FUNCTION_BLOCK Cylinder 
VAR_INPUT
END_VAR
VAR_OUTPUT
	bExtended : BOOL;
	bExtend : BOOL;
END_VAR
VAR
	fbExtendedSignal : BoolIn;
	fbExtend : BoolOut;
END_VAR

bExtended := fbExtendedSignal.getValue;
bExtend := fbExtend.getValue;

METHOD Extend : BOOL
VAR_INPUT
END_VAR
fbExtend.setValue := TRUE;
END_METHOD

PROPERTY getExtend : I_StepCondition
GET
getExtend := fbExtend;
END_GET
END_PROPERTY

METHOD Retract : BOOL
VAR_INPUT
END_VAR
fbExtend.setValue := FALSE;
END_METHOD

END_FUNCTION_BLOCK

(* stored: Version 1.1.0.1, ProductVersion 3.1.4024.2
   POU Cylinder: Id {4dff6417-8bf1-4724-a444-43bb6b5867e9}, SpecialFunc None
   Method Extend: Id {959ae6c2-4214-4061-b579-5b43c63e1617}
   Property getExtend: Id {551c2e8d-9793-498c-9e33-32fe5f29706c}
   Get Get: Id {70090b27-bd92-4955-9176-2f006b2ffbdc}
   Method Retract: Id {8f00f682-12a1-4f93-aad1-7d8e6b2d1427} *)
